FUNCTION_BLOCK Test_TExecution_SetErrorHandlesString_ErrorId EXTENDS T_UnitTestBase
VAR
    Execution : T_Execution;
END_VAR
VAR
    ErrorId : STRING := 'Custom error message';
END_VAR

{attribute 'analysis' := '-33'} // inhibit unused variable warning
METHOD RunTest
VAR
    ErrorMsg : STRING := 'Custom error message';
END_VAR
SUPER^.Init();

Execution.Start();
Execution.SetBusy();
Execution.SetError(ErrorMsg);

AssertIsTrue(Condition := Execution.ErrorMsg = 'Custom error message',
             Message   := 'Execution.ErrorMsg not correct');

TestCompleted := TRUE;
END_METHOD

END_FUNCTION_BLOCK

(* stored: Version 1.1.0.1, ProductVersion 3.1.4024.12
   POU Test_TExecution_SetErrorHandlesString_ErrorId: Id {16f08f29-068e-4798-90d6-e31f6569f288}, SpecialFunc None
   Method RunTest: Id {c802fc6f-c2eb-473d-9d52-1f1564e9b40b} *)
